{attribute 'qualified_only'}
VAR_GLOBAL CONSTANT
	MaxTestCount	  : DINT   := 50;
	MaxTestSuiteCount : DINT   := 10;
	DefaultPath		  : STRING := 'C:\ProgramData\Beckhoff\TwinCAT\3.1\Boot\TEST_Result.xml';
END_VAR

(* stored: Version 1.1.0.1
   GVL TestSuiteParameter: Id {71977508-7c74-4ec9-b7a4-3255aee38094}, ParameterList True *)
